// TIA Portal V16 export
// export: Created 2021-09-07T10:41:59.6924435Z, ExportSetting WithDefaults, DisplayName Totally Integrated Automation Portal, DisplayVersion V16 Update 3, DisplayName TIA Portal Version Control Interface, DisplayVersion V16 Update 2, DisplayName TIA Portal Openness, DisplayVersion V16 Update 3, DisplayName TIA Portal Teamcenter Gateway, DisplayVersion V16, DisplayName STEP 7 Professional, DisplayVersion V16 Update 3, DisplayName STEP 7 Safety, DisplayVersion V16, DisplayName WinCC Advanced, DisplayVersion V16 Update 3
ORGANIZATION_BLOCK "Main"   // OB1, LAD, ProgramCycle
TITLE = "Main Program Sweep (Cycle)"
{ S7_Optimized_Access := 'TRUE' }
VERSION : 0.1
// stored: AutoNumber true, IsIECCheckEnabled false, SetENOAutomatically false
   VAR_INPUT
      Initial_Call : Bool;   // Initial call of this OB
      Remanence : Bool;   // =True, if remanent data are available
   END_VAR
BEGIN

REGION Network 1
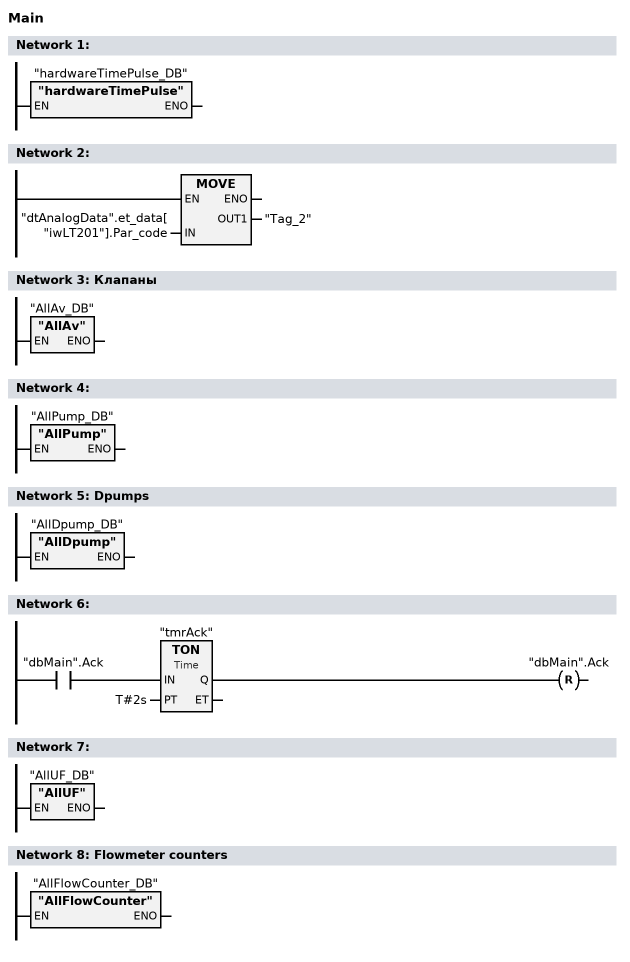
   RUNG wire#powerrail
      "hardwareTimePulse_DB"()
   END_RUNG
   // the same network as SCL:
   "hardwareTimePulse_DB"();   // "hardwareTimePulse"
END_REGION

REGION Network 2
   RUNG wire#powerrail
      Move(in := "dtAnalogData".et_data["iwLT201"].Par_code, out1 => "Tag_2")
   END_RUNG
   // the same network as SCL:
   "Tag_2" := "dtAnalogData".et_data["iwLT201"].Par_code;
END_REGION

REGION Network 3: Клапаны
   RUNG wire#powerrail
      "AllAv_DB"()
   END_RUNG
   // the same network as SCL:
   "AllAv_DB"();   // "AllAv"
END_REGION

REGION Network 4
   RUNG wire#powerrail
      "AllPump_DB"()
   END_RUNG
   // the same network as SCL:
   "AllPump_DB"();   // "AllPump"
END_REGION

REGION Network 5: Dpumps
   RUNG wire#powerrail
      "AllDpump_DB"()
   END_RUNG
   // the same network as SCL:
   "AllDpump_DB"();   // "AllDpump"
END_REGION

REGION Network 6
   RUNG wire#powerrail
      Contact( "dbMain".Ack )
      { S7_Templates := "time_type := Time" } "tmrAck".TON(pt := T#2s, et =>)
      R_Coil( "dbMain".Ack )
   END_RUNG
   // the same network as SCL:
   "tmrAck".TON(IN := "dbMain".Ack, PT := T#2s);
   IF "tmrAck".Q THEN "dbMain".Ack := FALSE; END_IF;
END_REGION

REGION Network 7
   RUNG wire#powerrail
      "AllUF_DB"()
   END_RUNG
   // the same network as SCL:
   "AllUF_DB"();   // "AllUF"
END_REGION

REGION Network 8: Flowmeter counters
   RUNG wire#powerrail
      "AllFlowCounter_DB"()
   END_RUNG
   // the same network as SCL:
   "AllFlowCounter_DB"();   // "AllFlowCounter"
END_REGION
END_ORGANIZATION_BLOCK
